FUNCTION_BLOCK FB_ReadParameterNC_TestDouble IMPLEMENTS  I_ReadParameter
VAR
    bError : BOOL;
    nErrorID : UDINT := 25000;
END_VAR

{warning 'Add property implementation'}
PROPERTY Aborted : BOOL
GET
END_GET
END_PROPERTY

{warning 'Add property implementation'}
PROPERTY Active : BOOL
GET
END_GET
END_PROPERTY

{warning 'Add property implementation'}
PROPERTY AmsNetID : T_AmsNetId
GET
END_GET
END_PROPERTY

{warning 'Add property implementation'}
PROPERTY AxisReadParamsInit : BOOL
GET
END_GET
END_PROPERTY

{warning 'Add property implementation'}
PROPERTY Busy : BOOL
GET
END_GET
END_PROPERTY

{warning 'Add property implementation'}
PROPERTY Done : BOOL
GET
END_GET
END_PROPERTY

{warning 'Add property implementation'}
PROPERTY EnInTargetTimeout : BOOL
GET
END_GET
END_PROPERTY

{warning 'Add property implementation'}
PROPERTY EnMaxSoftPosLimit : BOOL
GET
END_GET
END_PROPERTY

{warning 'Add property implementation'}
PROPERTY EnMinSoftPosLimit : BOOL
GET
END_GET
END_PROPERTY

{warning 'Add property implementation'}
PROPERTY EnPositionLagMonitoring : BOOL
GET
END_GET
END_PROPERTY

{warning 'Add property implementation'}
PROPERTY EnPositionRangeMonitoring : BOOL
GET
END_GET
END_PROPERTY

{warning 'Add property implementation'}
PROPERTY EnScaleFactorInternal : LREAL
GET
END_GET
END_PROPERTY

{warning 'Add property implementation'}
PROPERTY EnTargetPositionMonitoring : BOOL
GET
END_GET
END_PROPERTY

{warning 'Add property implementation'}
PROPERTY Error : BOOL
GET
Error := bError;
END_GET
SET
bError := Error;
END_SET
END_PROPERTY

{warning 'Add property implementation'}
PROPERTY ErrorID : UDINT
GET
ErrorId := nErrorID;
END_GET
SET
nErrorId := ErrorID;
END_SET
END_PROPERTY

{warning 'Add property implementation'}
PROPERTY InTargetTimeout : LREAL
GET
END_GET
END_PROPERTY

{warning 'Add property implementation'}
PROPERTY MaxPosLagFilterTime : LREAL
GET
END_GET
END_PROPERTY

{warning 'Add property implementation'}
PROPERTY MaxPosLagValue : LREAL
GET
END_GET
END_PROPERTY

{warning 'Add property implementation'}
PROPERTY MaxSoftPosLimit : LREAL
GET
END_GET
END_PROPERTY

{warning 'Add property implementation'}
PROPERTY Message : T_MAXSTRING
GET
END_GET
END_PROPERTY

{warning 'Add property implementation'}
PROPERTY MinSoftPosLimit : LREAL
GET
END_GET
END_PROPERTY

{warning 'Add property implementation'}
PROPERTY Port : WORD
GET
END_GET
END_PROPERTY

{warning 'Add property implementation'}
PROPERTY PositionRangeWindow : LREAL
GET
END_GET
END_PROPERTY

{warning 'Add method implementation '}
METHOD ReadParameters
VAR_INPUT
    Enable	: BOOL;
    RefreshDelay	: TIME;
END_VAR
END_METHOD

{warning 'Add property implementation'}
PROPERTY RefVeloSearch : LREAL
GET
END_GET
END_PROPERTY

{warning 'Add property implementation'}
PROPERTY RefVeloSync : LREAL
GET
END_GET
END_PROPERTY

{warning 'Add property implementation'}
PROPERTY TargetPositionMonitoringTime : LREAL
GET
END_GET
END_PROPERTY

{warning 'Add property implementation'}
PROPERTY TargetPositionWindow : LREAL
GET
END_GET
END_PROPERTY

END_FUNCTION_BLOCK

(* stored: Version 1.1.0.1
   POU FB_ReadParameterNC_TestDouble: Id {2d3a2979-0e7d-4c6e-bda2-88be2b8d08ba}, SpecialFunc None
   Property Aborted: Id {8474dbb5-4ab8-4e66-8860-ede44113b767}
   Get Get: Id {d7a4deed-1e3c-4686-bb9f-335ad5a82c0d}
   Property Active: Id {3177fe79-1c6c-40b1-9b72-4b3a9fa98b18}
   Get Get: Id {ba9aeebd-2459-4329-a455-498c49bb9a7b}
   Property AmsNetID: Id {13032c34-1a15-4c38-bae9-db218d73487c}
   Get Get: Id {a678eab7-7d12-4869-85b0-28f505eacd51}
   Property AxisReadParamsInit: Id {e9512799-3f3f-4cf6-9ae0-b09056cb6a95}
   Get Get: Id {d7fbc327-9208-4681-8395-d548536c2dc3}
   Property Busy: Id {813eb2f9-eff4-43c2-a176-fb7fa4f2a99c}
   Get Get: Id {83385d70-be19-437c-9e36-37f5bfbd406e}
   Property Done: Id {246aab87-a153-4441-bbb2-b12b7d5d43bd}
   Get Get: Id {f35d5fec-9278-40c8-955c-7aab2756eac8}
   Property EnInTargetTimeout: Id {a7f61ff7-0c72-4d94-9c9e-df55781cb77a}
   Get Get: Id {6fe02f44-3976-4577-ae4e-6a870cd94ca1}
   Property EnMaxSoftPosLimit: Id {03ac280f-5a51-4fdd-a9c8-5014b0cb14cb}
   Get Get: Id {ed0aff96-064a-4e39-9710-c8296f92cc4b}
   Property EnMinSoftPosLimit: Id {405a6593-958a-4507-93a9-569ba4fc10c7}
   Get Get: Id {3b85d3b5-d659-434d-93ed-8b274266dd87}
   Property EnPositionLagMonitoring: Id {93dc6b0b-40f1-46dc-966d-5191c84dea3f}
   Get Get: Id {87b0144f-036e-4962-8381-78791258ec4a}
   Property EnPositionRangeMonitoring: Id {bd2c1f49-c2f8-4ebe-acfd-5bace6d85466}
   Get Get: Id {1e6b0bf8-ab60-4b10-8d28-494b30b58d26}
   Property EnScaleFactorInternal: Id {a176806d-8507-419b-b721-5c9d6406d714}
   Get Get: Id {9ad45982-8ab6-475c-8aef-b61a77bdcb97}
   Property EnTargetPositionMonitoring: Id {1a409cb5-d3f6-4e48-9528-3698ad7320a2}
   Get Get: Id {9ae6d697-73aa-4788-95c0-818702f2a5f9}
   Property Error: Id {077f1294-4fda-4c92-947b-f0efec1090a9}
   Get Get: Id {c23e806c-962d-4265-8a9c-46bac8a84bbe}
   Set Set: Id {3394db00-42a8-484a-8e70-18f483daa069}
   Property ErrorID: Id {88e63353-f1c2-4014-b8f3-b964e67cad19}
   Get Get: Id {7b14065a-ef31-43b3-a378-40dd65b21057}
   Set Set: Id {19a1ee0e-e55c-423f-a491-ec1a205a499f}
   Property InTargetTimeout: Id {434627cd-e3f0-4755-a930-cc7f9d678a0a}
   Get Get: Id {f16a2042-b5b3-41c8-b119-2051ce916097}
   Property MaxPosLagFilterTime: Id {76cf887f-2e1c-4db0-82f5-95a3c1c3136f}
   Get Get: Id {ae6ec919-6c5f-4e41-8eb3-ecb359409279}
   Property MaxPosLagValue: Id {a2378202-3c6f-4d05-9af4-b5a132e0298c}
   Get Get: Id {415bf667-7ef5-46d4-a20d-4f40d660b100}
   Property MaxSoftPosLimit: Id {bd3bc724-5ea2-49fd-b158-19a5a1c24db3}
   Get Get: Id {20dfc5a4-68eb-4f26-a9f7-a912076fe365}
   Property Message: Id {0083a679-1b30-49eb-8a9d-7250ba3e50b8}
   Get Get: Id {d2df08c6-5dd5-488d-abfd-cb7add84465f}
   Property MinSoftPosLimit: Id {dcc2cf22-3191-48ab-94d9-d2da868287bb}
   Get Get: Id {dd55863c-359b-4ca8-bfc1-141972f3fb59}
   Property Port: Id {cb47a716-36ed-4586-af2c-5dadcb43d150}
   Get Get: Id {1a73d7bc-b168-4b46-bb23-87289c661558}
   Property PositionRangeWindow: Id {4dbc87d5-c7d6-42d6-a3e1-77c985e49e3e}
   Get Get: Id {fa16b1c4-4891-4c40-9f01-d1b4dc2f3df0}
   Method ReadParameters: Id {1f9bc1a5-7e1d-4e17-b037-a422a81fb0c0}
   Property RefVeloSearch: Id {8685362d-4da1-473a-97a8-a41259c76ece}
   Get Get: Id {a7a0629b-b85e-47bf-a435-42dfd49c4bdc}
   Property RefVeloSync: Id {698e5eaf-99fc-44fe-b03c-7e8a94ff9795}
   Get Get: Id {55bf763f-2959-45f8-bf1d-c5eef95f49f8}
   Property TargetPositionMonitoringTime: Id {3511b6c8-33aa-416c-8315-d8a5a7ad0193}
   Get Get: Id {6e2bc940-075f-43a6-9165-e4cc8a49dbcd}
   Property TargetPositionWindow: Id {1ead85dc-d5c2-4ca6-beca-21315b167273}
   Get Get: Id {fa14fe57-9392-43a4-a1c3-4005ca9017ac} *)
